// TIA Portal V17 export
FUNCTION "FC_风机燃气控制" : Void   // FC, LAD
{ S7_Optimized_Access := 'TRUE' }
   VAR_TEMP
      风机控制输出值 : Real;
      风压过渡 : Int;
   END_VAR
BEGIN
END_FUNCTION
